INTERFACE I_DirectoryEntry EXTENDS I_FileSystemEntry

END_INTERFACE

(* stored: Version 1.1.0.1, ProductVersion 3.1.4024.9
   Itf I_DirectoryEntry: Id {0f93bcd3-411b-4626-9e13-8828c5f6c9df} *)
